FUNCTION_BLOCK Demo 
VAR_INPUT
	
			DemoTable					: 			STRING(3); // Demo table type 
			bDpad_R						: 			BOOL;	// Dpad Right for starting the demo 
			bDpad_L						: 			BOOL; // Dpad Left to end demo 
			ReadyForDemo				: 			BOOL; // Handhske varible telling to start demo
			DemoStarting				:			BOOL; // Handshake to stop End Demo function
			StopEndFunction				:			BOOL; // Stop End function

END_VAR
VAR_OUTPUT
	
			RequestDemo					:			BOOL; // Handhske varible asking to start demo
			StartUserControl 			:			BOOL; // Varible to give user control of mover again

END_VAR
VAR

			TwoXOne 					:			TwoByOne; // Instacne of two by one demo
			FourXThree					:			FourByThree; // Instance of four by three demo	
			DemoStart					:			BOOL; // start the demo
			StopDemo					:			BOOL;
			
		
END_VAR


IF bDpad_R THEN //Link to Controller
	DemoStart := TRUE;
	StopDemo := FALSE;
END_IF

IF DemoStart THEN 
	RequestDemo := TRUE;
	IF ReadyForDemo THEN
		IF DemoTable = '2x1' THEN
			TwoXOne.Start := TRUE; 
		ELSIF DemoTable = '4x3' THEN
			FourXThree.Start := TRUE;
		ELSIF DemoTable = 'NaN' THEN
			//Do Nothing 
		END_IF
	END_IF
END_IF


IF bDpad_L THEN
	StopDemo := TRUE; 
	DemoStart := FALSE;
END_IF


IF StopDemo THEN 
	IF TwoXOne.Running OR FourXThree.Running THEN
		IF DemoTable = '2x1' THEN
			TwoXOne.Stop := TRUE; 
		ELSIF DemoTable = '4x3' THEN
			FourXThree.Stop := TRUE;
		ELSIF DemoTable = 'NaN' THEN
			//Do Nothing 
		END_IF
	END_IF
END_IF

IF 	TwoXOne.Stop AND FourXThree.Stop THEN
	StopDemo := FALSE;
	RequestDemo := FALSE;
	StartUserControl := TRUE;
	IF StopEndFunction THEN
		StartUserControl := FALSE;
	END_IF
END_IF

ACTION Cyclic:
FourXThree();
TwoXOne();
END_ACTION

METHOD EndDemo
VAR_INPUT
END_VAR
END_METHOD

METHOD StartDemo
VAR_INPUT
END_VAR
END_METHOD

END_FUNCTION_BLOCK

(* stored: Version 1.1.0.1, ProductVersion 3.1.4024.12
   POU Demo: Id {02e2345e-d9a2-4cec-9620-e2a4beef5936}, SpecialFunc None
   Action Cyclic: Id {0311b125-da15-4b48-bc76-7579ce2660fd}
   Method EndDemo: Id {6854c3e9-f245-4ca4-a051-8800377238fb}
   Method StartDemo: Id {db17a7a0-a8fd-475e-8ecc-aae4bf70183f} *)
